FUNCTION DEAD_ZONE (* dead_zone2 is a linear transfer function which follows a linear function except for x is close to 0. *)
  (* Standard: 61499-1 *)
  (* Version 1.0, 2025-12-19, Franz Höpfinger *)
  PACKAGE OSCAT::Basic::POUs::Engineering::Control;
  IMPORT eclipse4diac::core::TypeHash;
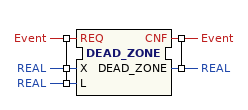
  EVENT_INPUT
    REQ WITH X, L;
  END_EVENT
  EVENT_OUTPUT
    CNF WITH DEAD_ZONE;
  END_EVENT
  VAR_INPUT
    X : REAL;
    L : REAL;
  END_VAR
  VAR_OUTPUT
    DEAD_ZONE : REAL;
  END_VAR
  BODY IN ST:
PACKAGE OSCAT::Basic::POUs::Engineering::Control;

(* dead_zone2 is a linear transfer function which follows a linear function except for x is close
 * to 0. *)
FUNCTION DEAD_ZONE : REAL
VAR_INPUT
	X : REAL;
	L : REAL;
END_VAR

(*
 * version 1.2	11. mar. 2009 programmer 	hugo tested by		oscat
 * *
 * dead_zone2 is a linear transfer function which follows a linear function except for x is close to
 * 0.
 * Y = X if abs(x) > L otherwise its 0.
 *)
IF ABS(X) > L THEN
	DEAD_ZONE := X;
ELSE
	DEAD_ZONE := 0.0;
END_IF;

END_FUNCTION

(* revision history hm	12. feb. 2007	rev 1.0 original version
 * *
 * hm	14. jun. 2008	rev 1.1 improved performance
 * *
 * hm	11. mar. 2009	rev 1.2 real constants updated to new systax using dot *)
  END_BODY
END_FUNCTION
